(* CODESYS project chemical-mixer.project
   Title: projekt
   Version: 0.0.0.0
   Author: jasar

Project tree, tasks and I/O mapping:
  MyController : TM238LDD24DT, Schneider Electric, order no. TM238LDD24DT, version 4.0.1.28
      settings: OpcUa Enable = False
    application Application
      task MAST (cyclic, interval 20 ms, priority 15, watchdog 100 ms x 1) calls POU
      task Task (cyclic, interval t#20ms, priority 16) calls POU_1
      task Task_1 (cyclic, interval t#10ms, priority 1) calls POU_2
      global variables GVL
      program POU [FBD]
      program POU_1 [ST]
      Symbols
      program POU_2 [ST]
    Embedded Functions
      IO : IO, Schneider Electric, version 4.0.1.28
          input  iwIO_IW0 : WORD  // IW0
          output qwIO_QW0 : WORD  // QW0
      HSC : HSC, Schneider Electric, version 4.0.1.28
      PTO_PWM : PTO_PWM, Schneider Electric, version 4.0.1.28
    Serial Line
      SoMachine_Network_Manager : SoMachine-Network Manager, Schneider Electric, version 4.0.0.2
  HMIS5T : HMIS5T, Schneider Electric, order no. HMIS5T, version 3.5.3.54
    HMI Application
    Ethernet
      SoMachine_Network_Manager2 : SoMachine-Network Manager, Schneider Electric, version 4.0.0.2
    COM1
      SoMachine_Network_Manager1 : SoMachine-Network Manager, Schneider Electric, version 4.0.0.2
    USB
      SoMachine_Network_Manager3 : SoMachine-Network Manager, Schneider Electric, version 4.0.0.2
  Vijeo Designer Project Container Data
  Vijeo Designer Project Container
*)

// MyController/Application/GVL
VAR_GLOBAL
	termicka_mikser: BOOL;
	termicka_pumpa: BOOL;
	greska_senzor_B0: BOOL;
	greska_senzor_B1: BOOL;
	greska_senzor_B2: BOOL;
	greska_senzor_B3: BOOL;
	greska_senzor_B4: BOOL;
	pomocna_iskljuci: BOOL;
	prebaci_panel3_: BOOL;
	brojac: INT;
	senzor_B5_: BOOL;
	senzor_B4_: BOOL;
	senzor_B3_: BOOL;
	senzor_B2_: BOOL;
	senzor_B1_: BOOL;
	senzor_B0_: BOOL;
END_VAR

// MyController/Application/POU
PROGRAM POU
VAR
	taster_S3: BOOL;
	rezervoar1: RS;
	rezervoar2: RS;
	rezervoar3: RS;
	rezervoar4: RS;
	rezervoar5: RS;
	svjetlosni_signal_H0: RS;
	svjetlosni_signal_H1: RS;
	mjesalica: RS;
	pumpa: RS;
	iskljucenje_mjesalice: TP;
	Q_ventil_1: BOOL;
	Q_ventil_2: BOOL;
	Q_ventil1_3: BOOL;
	Q_ventil1_4: BOOL;
	Q_ventil1_5: BOOL;
	Q_mjesalica: BOOL;
	Q_pumpa: BOOL;
	Q_lampica_H1: BOOL;
	Q_lampica_H0: BOOL;
	F_TRIG_iskljucenje_mjesalice: F_TRIG;
	iskljuci_mjesalicu: BOOL;
	F_TRIG_taster_S2: F_TRIG;
	F_TRIG_taster_S0: F_TRIG;
	iskljuci_sistem: BOOL;
	zaustavi_mjesalicu: BOOL;
	senzor_B5: BOOL;
	senzor_B1: BOOL;
	senzor_B2: BOOL;
	senzor_B3: BOOL;
	senzor_B4: BOOL;
	taster_S2: BOOL;
	taster_S0: BOOL;
	taster_S1: BOOL;
	R_TRIG_taster_S2: R_TRIG;
	SR_mjesalica: SR;
	taster_S4: BOOL;
	senzor_B0: BOOL;
	SR_lampica_H0: SR;
	zaustavljanje_mjesalice: RS;
	iskljucenje_sistema: RS;
	F_TRIG_taster_S0_mjesalica: F_TRIG;
	F_TRIG_taster_S2_mjesalica: F_TRIG;
	F_TRIG_taster_S0_lampica_H0: F_TRIG;
	iskljucenje_ventila_0: TP;
	F_TRIG_iskljucenje_ventila_0: F_TRIG;
	iskljuci_ventil_0: BOOL;
	ventil_0: RS;
	Q_ventil_0: BOOL;
	svjetlosni_signal_H1_: SR;
	prebaci_panel3: BOOL;
	pomocni_r_trig: R_TRIG;
	pomocni_f_trig: F_TRIG;
	rezervoar1_: SR;
END_VAR

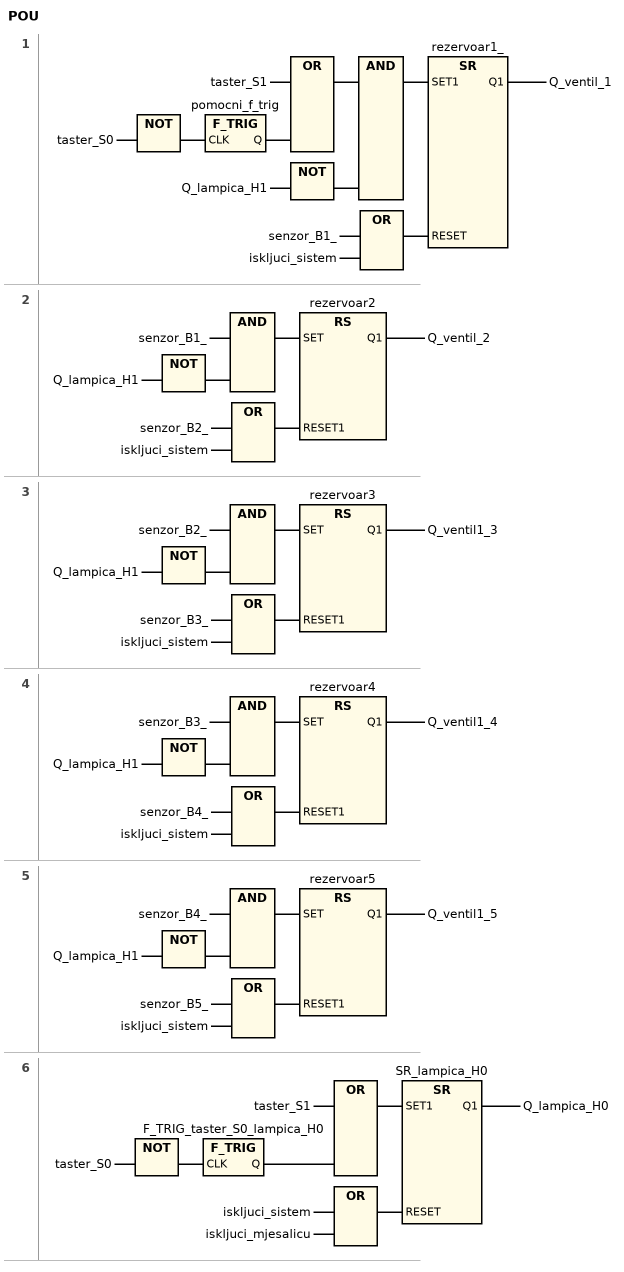
// NETWORK 1
pomocni_f_trig(CLK := NOT taster_S0); // F_TRIG
rezervoar1_(SET1 := (taster_S1 OR pomocni_f_trig.Q) AND NOT Q_lampica_H1, RESET := senzor_B1_ OR iskljuci_sistem); // SR
Q_ventil_1 := rezervoar1_.Q1;

// NETWORK 2
rezervoar2(SET := senzor_B1_ AND NOT Q_lampica_H1, RESET1 := senzor_B2_ OR iskljuci_sistem); // RS
Q_ventil_2 := rezervoar2.Q1;

// NETWORK 3
rezervoar3(SET := senzor_B2_ AND NOT Q_lampica_H1, RESET1 := senzor_B3_ OR iskljuci_sistem); // RS
Q_ventil1_3 := rezervoar3.Q1;

// NETWORK 4
rezervoar4(SET := senzor_B3_ AND NOT Q_lampica_H1, RESET1 := senzor_B4_ OR iskljuci_sistem); // RS
Q_ventil1_4 := rezervoar4.Q1;

// NETWORK 5
rezervoar5(SET := senzor_B4_ AND NOT Q_lampica_H1, RESET1 := senzor_B5_ OR iskljuci_sistem); // RS
Q_ventil1_5 := rezervoar5.Q1;

// NETWORK 6
F_TRIG_taster_S0_lampica_H0(CLK := NOT taster_S0); // F_TRIG
SR_lampica_H0(SET1 := taster_S1 OR F_TRIG_taster_S0_lampica_H0.Q, RESET := iskljuci_sistem OR iskljuci_mjesalicu); // SR
Q_lampica_H0 := SR_lampica_H0.Q1;

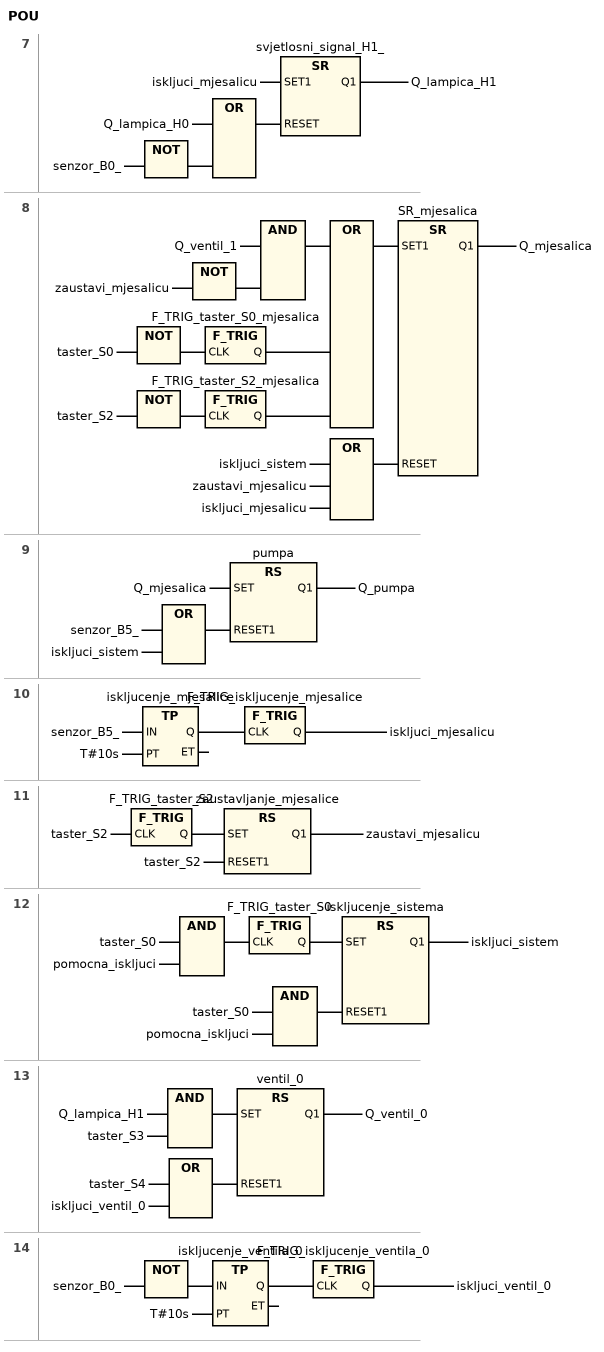
// NETWORK 7
svjetlosni_signal_H1_(SET1 := iskljuci_mjesalicu, RESET := Q_lampica_H0 OR NOT senzor_B0_); // SR
Q_lampica_H1 := svjetlosni_signal_H1_.Q1;

// NETWORK 8
F_TRIG_taster_S0_mjesalica(CLK := NOT taster_S0); // F_TRIG
F_TRIG_taster_S2_mjesalica(CLK := NOT taster_S2); // F_TRIG
SR_mjesalica(SET1 := Q_ventil_1 AND NOT zaustavi_mjesalicu OR F_TRIG_taster_S0_mjesalica.Q OR F_TRIG_taster_S2_mjesalica.Q, RESET := iskljuci_sistem OR zaustavi_mjesalicu OR iskljuci_mjesalicu); // SR
Q_mjesalica := SR_mjesalica.Q1;

// NETWORK 9
pumpa(SET := Q_mjesalica, RESET1 := senzor_B5_ OR iskljuci_sistem); // RS
Q_pumpa := pumpa.Q1;

// NETWORK 10
iskljucenje_mjesalice(IN := senzor_B5_, PT := T#10s); // TP
F_TRIG_iskljucenje_mjesalice(CLK := iskljucenje_mjesalice.Q); // F_TRIG
iskljuci_mjesalicu := F_TRIG_iskljucenje_mjesalice.Q;

// NETWORK 11
F_TRIG_taster_S2(CLK := taster_S2); // F_TRIG
zaustavljanje_mjesalice(SET := F_TRIG_taster_S2.Q, RESET1 := taster_S2); // RS
zaustavi_mjesalicu := zaustavljanje_mjesalice.Q1;

// NETWORK 12
F_TRIG_taster_S0(CLK := taster_S0 AND pomocna_iskljuci); // F_TRIG
iskljucenje_sistema(SET := F_TRIG_taster_S0.Q, RESET1 := taster_S0 AND pomocna_iskljuci); // RS
iskljuci_sistem := iskljucenje_sistema.Q1;

// NETWORK 13
ventil_0(SET := Q_lampica_H1 AND taster_S3, RESET1 := taster_S4 OR iskljuci_ventil_0); // RS
Q_ventil_0 := ventil_0.Q1;

// NETWORK 14
iskljucenje_ventila_0(IN := NOT senzor_B0_, PT := T#10s); // TP
F_TRIG_iskljucenje_ventila_0(CLK := iskljucenje_ventila_0.Q); // F_TRIG
iskljuci_ventil_0 := F_TRIG_iskljucenje_ventila_0.Q;

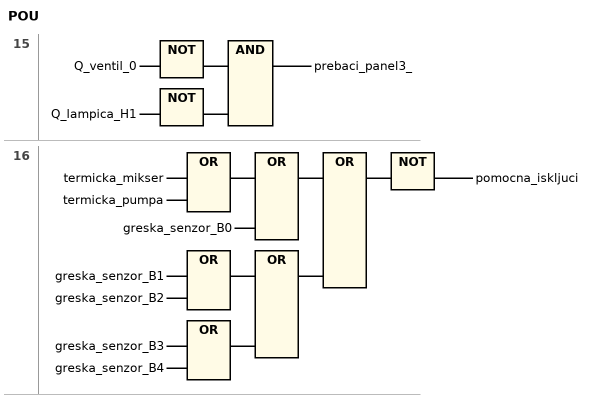
// NETWORK 15
prebaci_panel3_ := NOT Q_ventil_0 AND NOT Q_lampica_H1;

// NETWORK 16
pomocna_iskljuci := NOT (((termicka_mikser OR termicka_pumpa) OR greska_senzor_B0) OR ((greska_senzor_B1 OR greska_senzor_B2) OR (greska_senzor_B3 OR greska_senzor_B4)));

END_PROGRAM

// MyController/Application/POU_1
PROGRAM POU_1
VAR
END_VAR


IF senzor_B5_ = TRUE THEN
	brojac := 6;
ELSIF senzor_B4_ = TRUE THEN
	brojac := 5;
ELSIF senzor_B3_ = TRUE THEN
	brojac := 4;
ELSIF senzor_B2_ = TRUE THEN
	brojac := 3;
ELSIF senzor_B1_ = TRUE THEN
	brojac := 2;
ELSIF senzor_B0_ = TRUE THEN
	brojac := 1;
ELSE
	brojac := 0;
END_IF

END_PROGRAM

// MyController/Application/POU_2
PROGRAM POU_2
VAR
END_VAR

IF ( senzor_B5_ OR senzor_B4_ OR senzor_B3_ OR senzor_B2_ OR senzor_B1_ ) AND senzor_B0_ = FALSE THEN
	greska_senzor_B0 := TRUE;
ELSE
	greska_senzor_B0 := FALSE;
END_IF

IF ( senzor_B5_ OR senzor_B4_ OR senzor_B3_ OR senzor_B2_ ) AND senzor_B1_ = FALSE THEN
	greska_senzor_B1 := TRUE;
ELSE
	greska_senzor_B1 := FALSE;
END_IF

IF ( senzor_B5_ OR senzor_B4_ OR senzor_B3_ ) AND senzor_B2_ = FALSE THEN
	greska_senzor_B2 := TRUE;
ELSE
	greska_senzor_B2 := FALSE;
END_IF

IF ( senzor_B5_ OR senzor_B4_ ) AND senzor_B3_ = FALSE THEN
	greska_senzor_B3 := TRUE;
ELSE
	greska_senzor_B3 := FALSE;
END_IF

IF ( senzor_B5_ ) AND senzor_B4_ = FALSE THEN
	greska_senzor_B4 := TRUE;
ELSE
	greska_senzor_B4 := FALSE;
END_IF

END_PROGRAM
